{library PRIVATE}
(*
  Private Funtcion:
  Decode Status information messages.

*)
FUNCTION _GetStatusInformation : StatusInformationData
VAR_INPUT
	Data: 				DataGram;
END_VAR
VAR
END_VAR

_GetStatusInformation.Progress:=DWORD_TO_INT((SHR(Data.ParameterDW, 24) AND  16#FF));
_GetStatusInformation.FunctionNumber:=BYTE_TO_INT(Data.FunctionNumber);
_GetStatusInformation.ReturnValue:=BYTE_TO_INT(Data.FunctionType);
_GetStatusInformation.Extra:=BYTE_TO_INT(Data.ParameterB);

END_FUNCTION

(* stored: Version 1.1.0.1, ProductVersion 3.1.4022.12
   POU _GetStatusInformation: Id {5ab44f4b-f737-4fae-8cbe-d3fa9859db8c}, SpecialFunc None *)
